// Mitsubishi GX Works2 project: helloword 2709   PLC: Q03UDV

PROGRAM MAIN
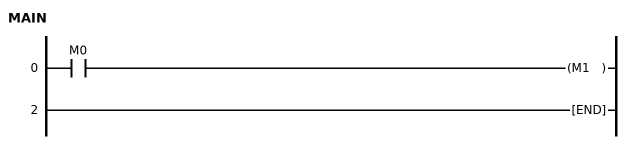
0     LD      M0
      OUT     M1
2     END
END_PROGRAM
